# EPICS substitutions: old/bl6-SkfChopper/bl6-SkfChopperApp/Db/skf2_saveRst.substitutions
file save_restoreStatus.db
{
pattern {P}
       {BL6:SavRst:ChopSkf2:}
}
